{attribute 'GeneratedUsingTerminal: EL6080-0000-0016'}
{attribute addProperty BoxType "EL6080-0000-0016"}
{attribute addProperty Id "ControlAT %Q*ARRAY [0..1] OF USINT0"}
{attribute addProperty CRC "2284853588"}
{attribute addProperty Size "0"}
TYPE Control_88301954 EXTENDS OutputBase_10CEE7DE :
STRUCT
	{attribute addProperty Name "Control"}
	Control AT %Q* : ARRAY [0..1] OF USINT;
END_STRUCT
END_TYPE

(* stored: Version 1.2.0.0, ProductVersion 3.1.4024.9
   DUT Control_88301954: Id {541d2d1b-5dbf-47a6-b1e3-3b46584715b7} *)
